# EPICS substitutions: IsoPlaneApp/Db/IsoPlane.substitutions
file "db/IsoPlane.template"
{
    pattern{P, R, PORT}
    {"WIZZLERHD:HZDR:", "IsoPlane:", "IsoPlane"}
}
